// TIA Portal V18 export
VAR_GLOBAL   // PLC tag table "Type"
   iSSP1p AT %I0.0 : Bool;
   iSSP1 AT %I0.1 : Bool;
   iSSP2p AT %I0.2 : Bool;
   iSSP2 AT %I0.3 : Bool;
   oSSP1t1 AT %Q17.2 : Bool;
   oSSP1t2 AT %Q17.3 : Bool;
   oSSP2t1 AT %Q17.4 : Bool;
   oSSP2t2 AT %Q17.5 : Bool;
END_VAR
